(* IEC 61131-3 sources: moqui-plc/simatic-ax/src/moqui/runtime/component/mantle-hvac/src/main/org/moqui/device, 5 files *)

(* ---- AirDistributionControllerStatus.st ---- *)
TYPE AirDistributionControllerStatus : (
    Init,
    HighPhase,
    TransitionToLow,
    LowPhase,
    TransitionToHigh
); END_TYPE

(* ---- DeviceFacade.st ---- *)
(*
 * DeviceFacade implementation for managing devices and logical parameters.
 *
 * Naming rules:
 *   deviceName + parameterName or parameterName -> logical signal
 *   deviceName + parameterName or parameterName + Min/Max -> limits
 *
 * All digital signals (boolean) are active-high (positive logic).
 * All durations are expressed in seconds TUnit.
 *)
TYPE DeviceFacade : STRUCT
	(* HVAC process control parameters (setpoints, limits, etc.) and process sensor signals *)
    (* Cell T+RH sensor  *)
    (* Setpoints and limits - mapped from recipe *)
    tempSetpoint : REAL; (* °C target process temperature *)
    tempHysteresis : REAL; (* °C symmetric hysteresis band *)
    tempMin : REAL;   (* °C absolute lower limit (alarm) *)
    tempMax : REAL; (* °C absolute upper limit (alarm) *)
    rhSetpoint : REAL; (* %  target relative humidity *)
    rhHysteresis : REAL; (* %  symmetric hysteresis band *)
    rhMin : REAL; (* % lower limit *)
    rhMax : REAL; (* % upper limit *)
    (* Feedback - wired from InputSignalUpdate each scan *)
    tempFeedback : REAL; (* °C zone air temperature *)
    rhFeedback : REAL; (* % zone relative humidity *)

    (* Duct T+RH sensor (probe in the pipes) *)
    (* Limits - mapped from recipe or fixed commissioning values *)
    ductTempMin : REAL; (* °C minimum safe supply-air temperature *)
    ductTempMax : REAL; (* °C maximum safe supply-air temperature *)
    ductRhMax : REAL; (* % maximum allowed supply-air humidity *)
    (* Feedback - wired from InputSignalUpdate each scan *)
    ductTempFeedback : REAL; (* °C supply-air temperature in duct *)
    ductRhFeedback : REAL; (* % supply-air relative humidity in duct *)

    (* Boolean predicates - computed each scan by MainRuleEngine *)
    (* Cell sensor *)
    tempInRange : BOOL; (* tempMin+hys <= T <= tempMax-hys *)
    tempAtSetpoint : BOOL; (* |T - Tsp| <= hys *)
    tempAboveSetpointBand : BOOL; (* T >= tempSetpoint + tempHysteresis *)
    tempBelowSetpointBand : BOOL; (* T <= tempSetpoint - tempHysteresis *)
    tempOverMax : BOOL; (* T > tempMax *)
    tempOverMin : BOOL; (* T > tempMin *)
    tempUnderMin : BOOL; (* T < tempMin *)
    tempUnderMax : BOOL; (* T < tempMax *)
    rhAtSetpoint : BOOL;
    rhOverMax  : BOOL; (* RH > rhMax - hys *)
    rhUnderMin : BOOL; (* RH < rhMin + hys *)
    rhOverMin : BOOL;
    rhUnderMax : BOOL;
    (* Duct sensor - safety predicates *)
    ductTempOverMax : BOOL; (* Supply air too hot -> temperature limit violation *)
    ductTempUnderMin : BOOL; (* Supply air too cold -> temperature limit violation *)
    ductRhOverMax : BOOL; (* Supply air saturated -> condensation risk *)

    (* Operating-mode flags and process timing (mapped from recipe). *)
    rhControlEnabled : BOOL; (* Cooling+Heating both active for RH ctrl *)
    rhControlOnly : BOOL; (* Stop when RH <= rhMin regardless of time *)
    (* Air mixing *)
    airMixingEnabled : BOOL;
    airMixingFanEnableRequest : BOOL;
    airMixingFanDisableRequest : BOOL;
    airMixingFan : Actuator;
	(* Air distribution setpoints *)
	airDistributionEnabled : BOOL;
    setPointTimeHigh : UINT; (* Required cumulative time for high throw [s] *)
    setPointTimeLow : UINT; (* Required cumulative time for low throw [s] *)
    (* Process cycle durations (seconds) *)
    processEstimatedDuration : UDINT;
    processMinDuration : UDINT;
    processActualDuration : UDINT;
    processRemainingDuration : UDINT;
    (* Process time tracking *)
    (* Run / break cycle - Mode E *)
    estimatedRuntime : UDINT;
    minRuntime : UDINT;
    actualRuntime : UDINT;
    estimatedBreakDuration : UDINT;
    minBreakDuration : UDINT;
    actualBreakDuration : UDINT;
    (* Flags *)
    timeBreakEnabled : BOOL; (* TRUE while in break period *)
    isCompleted : BOOL; (* TRUE when the work effort is finished *)

    (* Main FSM state and transition request/acknowledge commands *)
    status : MainStatus := MainStatus#Standby;
    lastStatus : MainStatus := MainStatus#Standby;
    (*
     * Internally generated transition requests (set by MainRuleEngine,
     * consumed and cleared by Main.pou each scan)
     *)
    standbyRequest : BOOL;
    ventilationRequest : BOOL;
    coolingRequest : BOOL;
    heatingRequest : BOOL;
    dryingRequest : BOOL;
    faultRequest : BOOL;
    resetRequest : BOOL;

    (* HVAC devices *)

    (* Cold glycol group *)
    (* Enable/disable requests: written by Main component, read by DeviceManager *)
    coldGroupEnableRequest : BOOL;
    coldGroupDisableRequest : BOOL;
    (* Glycol circulating pump - on/off Actuator *)
    coldGlycolPump : Actuator;
    (* Modulating glycol valve - continuous PID control *)
    coldGlycolValve : ProcessPid;

    (* Hot glycol group *)
    hotGroupEnableRequest : BOOL;
    hotGroupDisableRequest : BOOL;
    hotGlycolPump : Actuator;
    hotGlycolValve : ProcessPid;

    (* AHU fan *)
    ahuFanEnableRequest : BOOL;
    (* Speed setpoint (0.0 … 100.0 %) - from recipe *)
    ahuFanSpeedSetpoint : REAL;
    (* Speed feedback (0.0 … 100.0 %) - from InputSignalUpdate *)
    ahuFanSpeedFeedback : REAL;
    ahuFan : ProcessPid;

    (* Air-flow distributor *)
    (* Treated as Actuator with additional ref/feedback.
     * The drive alternates air distribution between left and right ducts.
     * ref = time-split setpoint (0-100 %, 0 = full left, 100 = full right).
     * feedback = actual drive speed feedback.
	 *)
    airFlowEnableRequest : BOOL;
    airFlowDisableRequest : BOOL;
    airFlowRef : REAL; (* duty-cycle / distribution setpoint *)
    airFlowSpeedFeedback : REAL; (* drive speed feedback *)
    airFlow : Actuator;

    (* High flow damper *)
    highFlowDamperEnableRequest : BOOL;
    highFlowDamperDisableRequest : BOOL;
    highFlowDamper : Actuator;

    (* Low flow damper *)
    lowFlowDamperEnableRequest : BOOL;
    lowFlowDamperDisableRequest : BOOL;
    lowFlowDamper : Actuator;

    (* Signal management - centralised fault / alarm / warning engine *)
    signalMgmt : SignalMgmt;
END_STRUCT; END_TYPE

(* ---- AirDistributionController.st ---- *)
(*
 * AirDistributionController: Logical sequencer for alternating high/low air throw.
 *
 * Implements cumulative timing logic for throw phases:
 * - Time advances only during active operation (operationType = Run AND enable = TRUE).
 * - Counters are frozen (retained) during standby/pause phases.
 * - Implements a Make-Before-Break transition between ducts to prevent overpressure peaks,
 * leveraging the asynchronous handshake mechanism (VAR_IN_OUT) of the underlying Actuator instances.
 *)
FUNCTION_BLOCK AirDistributionController
	VAR_EXTERNAL
	    dev : DeviceFacade;
	END_VAR
	VAR_INPUT
	    operationType : OperatingMode := OperatingMode#Init;
	    enable : BOOL; (* Local run permission (e.g., air flow running + air mixing enabled) *)
	    clock1s : BOOL; (* 1-second base clock pulse *)
	END_VAR
	VAR CONSTANT
	    componentName : STRING := 'HVAC_AIR_GROUP';
	END_VAR
	VAR
		(* Logger facade *)
	    logger : LoggerFacade;
	    status : AirDistributionControllerStatus := AirDistributionControllerStatus#Init;
	    cumulatedTimeHigh : UINT := UINT#0;
	    cumulatedTimeLow : UINT := UINT#0;
	END_VAR

	(* Logger facade init *)
	logger.enable := TRUE; logger.loggerName := componentName;

	(* Initialization or reset upon critical Stop *)
	IF operationType = OperatingMode#Init THEN
	    logger(message := 'Init air distribution controller.', level := LogLevel#DEBUG);
	    status := AirDistributionControllerStatus#Init;
	    cumulatedTimeHigh := UINT#0;
	    cumulatedTimeLow := UINT#0;
		dev.highFlowDamperEnableRequest := TRUE;
		dev.highFlowDamperDisableRequest := FALSE;
		dev.lowFlowDamperEnableRequest := FALSE;
		dev.lowFlowDamperDisableRequest := TRUE;
	    RETURN;
	END_IF;

	(* Logic advances ONLY if the system is in Run mode and local enable is active *)
	IF (operationType = OperatingMode#Run) AND enable THEN

	    CASE status OF

	        AirDistributionControllerStatus#Init:
	            (* Startup sequence: defaults to the high throw phase *)
	            dev.highFlowDamperEnableRequest := TRUE;
	 		   	dev.highFlowDamperDisableRequest := FALSE;
	            dev.lowFlowDamperEnableRequest := FALSE;
	 		   	dev.lowFlowDamperDisableRequest := TRUE;
	            logger(message := 'Enter high throw phase.', level := LogLevel#DEBUG);
	            status := AirDistributionControllerStatus#HighPhase;

	        AirDistributionControllerStatus#HighPhase:
	            (* Advance cumulative timer *)
	            IF clock1s THEN
	                cumulatedTimeHigh := cumulatedTimeHigh + UINT#1;
	            END_IF;

	            (* Evaluate switching threshold *)
	            IF dev.setPointTimeHigh > UINT#0 AND cumulatedTimeHigh >= dev.setPointTimeHigh THEN
	                cumulatedTimeHigh := UINT#0;
	                (* Make-Before-Break Interlock / Asynchronous Handshake *)
					dev.highFlowDamperEnableRequest := FALSE;
					dev.highFlowDamperDisableRequest := TRUE;
					dev.lowFlowDamperEnableRequest := TRUE;
					dev.lowFlowDamperDisableRequest := FALSE;
	                logger(message := 'Transition to low throw.', level := LogLevel#DEBUG);
	                status := AirDistributionControllerStatus#TransitionToLow;
	            END_IF;

	        AirDistributionControllerStatus#TransitionToLow:
	            (* * Monitor the falling edge of the request signals.
	             * The Actuator block internally clears the VAR_IN_OUT variable once
	             * the physical maneuver is completed. This ensures the sequencer
	             * advances only after the hardware has reached its target position.
	             *)
	            IF NOT dev.highFlowDamperDisableRequest AND NOT dev.lowFlowDamperEnableRequest THEN
	                logger(message := 'Enter low throw phase.', level := LogLevel#DEBUG);
	                status := AirDistributionControllerStatus#LowPhase;
	            END_IF;

	        AirDistributionControllerStatus#LowPhase:
	            (* Advance cumulative timer *)
	            IF clock1s THEN
	                cumulatedTimeLow := cumulatedTimeLow + UINT#1;
	            END_IF;

	            (* Evaluate switching threshold *)
	            IF dev.setPointTimeLow > UINT#0 AND cumulatedTimeLow >= dev.setPointTimeLow THEN
	                cumulatedTimeLow := UINT#0;
	                (* Make-Before-Break Interlock / Asynchronous Handshake *)
					dev.highFlowDamperEnableRequest := TRUE;
					dev.highFlowDamperDisableRequest := FALSE;
					dev.lowFlowDamperEnableRequest := FALSE;
					dev.lowFlowDamperDisableRequest := TRUE;
	                logger(message := 'Transition to high throw.', level := LogLevel#DEBUG);
	                status := AirDistributionControllerStatus#TransitionToHigh;
	            END_IF;

	        AirDistributionControllerStatus#TransitionToHigh:
	            (* Wait for hardware positioning confirmation *)
	            IF NOT dev.lowFlowDamperDisableRequest AND NOT dev.highFlowDamperEnableRequest THEN
	                logger(message := 'Enter high throw phase.', level := LogLevel#DEBUG);
	                status := AirDistributionControllerStatus#HighPhase;
	            END_IF;
	    END_CASE;
	ELSE
	    (* Standby / Pause Condition *)
	    (*
	     * During standby (OperatingMode#Standby OR enable = FALSE), the FB does
	     * not increment any timers. The current status and Request variables are
	     * frozen, maintaining the hardware in its last consolidated stable state.
	     *)
	    ;
	END_IF;
	END_FUNCTION_BLOCK

(* ---- DeviceDiagnostics.st ---- *)
(* Device diagnostics *)
FUNCTION_BLOCK DeviceDiagnostics
	VAR_EXTERNAL
		dev : DeviceFacade;
	END_VAR
	VAR_INPUT
		operationType : OperatingMode := OperatingMode#Run;
	END_VAR
	VAR_OUTPUT
		error : BOOL;
	END_VAR

	error := TRUE;

	(* Signal management engine *)
	(*
	 * Prepare a fresh scan (clears the accumulated output action).
	 * Then process each device signal in priority order.
	 * ImmediateStop -> faultRequest := TRUE -> Main enters Fault state.
	 *)
	dev.signalMgmt(operationType := SignalMgmtOperatingMode#Prepare);
	dev.signalMgmt.operationType := SignalMgmtOperatingMode#Process;

	(* Device faults *)
	dev.signalMgmt(
		loggerName := dev.ahuFan.loggerName,
		code := 16#0001,
		category := SignalCategory#Alarm,
		resetPol := ResetPolicy#UnconditionedReset,
		activationCondition := dev.ahuFan.invalidConfig,
		outputAction := DWORD#16#0002);
	dev.signalMgmt(
		loggerName := dev.airFlow.loggerName,
		code := 16#0002,
		category := SignalCategory#Alarm,
		resetPol := ResetPolicy#UnconditionedReset,
		activationCondition := dev.airFlow.fault,
		outputAction := DWORD#16#0002);
	dev.signalMgmt(
		loggerName := dev.coldGlycolPump.loggerName,
		code := 16#0003,
		category := SignalCategory#Alarm,
		resetPol := ResetPolicy#UnconditionedReset,
		activationCondition := dev.coldGlycolPump.fault,
		outputAction := DWORD#16#0002);
	dev.signalMgmt(
		loggerName := dev.coldGlycolValve.loggerName,
		code := 16#0004,
		category := SignalCategory#Alarm,
		resetPol := ResetPolicy#UnconditionedReset,
		activationCondition := dev.coldGlycolValve.invalidConfig,
		outputAction := DWORD#16#0002);
	dev.signalMgmt(
		loggerName := dev.hotGlycolPump.loggerName,
		code := 16#0005,
		category := SignalCategory#Alarm,
		resetPol := ResetPolicy#UnconditionedReset,
		activationCondition := dev.hotGlycolPump.fault,
		outputAction := DWORD#16#0002);
	dev.signalMgmt(
		loggerName := dev.hotGlycolValve.loggerName,
		code := 16#0006,
		category := SignalCategory#Alarm,
		resetPol := ResetPolicy#UnconditionedReset,
		activationCondition := dev.hotGlycolValve.invalidConfig,
		outputAction := DWORD#16#0002);
	dev.signalMgmt(
		loggerName := dev.highFlowDamper.loggerName,
		code := 16#0007,
		category := SignalCategory#Alarm,
		resetPol := ResetPolicy#UnconditionedReset,
		activationCondition := dev.highFlowDamper.fault,
		outputAction := DWORD#16#0002);
	dev.signalMgmt(
		loggerName := dev.lowFlowDamper.loggerName,
		code := 16#0008,
		category := SignalCategory#Alarm,
		resetPol := ResetPolicy#UnconditionedReset,
		activationCondition := dev.lowFlowDamper.fault,
		outputAction := DWORD#16#0002);

	(*
	 * Duct safety alarms - supply-air temperature limits (ImmediateStop).
	 * Air that is too hot or too cold entering the curing room can damage
	 * or contaminate the product. These alarms are always evaluated
	 * regardless of the current FSM state.
	 *)
	dev.signalMgmt(
		loggerName := 'HVAC_DEMO_PLC',
		code := 16#0010,
		category := SignalCategory#Alarm,
		resetPol := ResetPolicy#UnconditionedReset,
		activationCondition := dev.ductTempOverMax,
		outputAction := DWORD#16#0002);
	dev.signalMgmt(
		loggerName := 'HVAC_DEMO_PLC',
		code := 16#0011,
		category := SignalCategory#Alarm,
		resetPol := ResetPolicy#UnconditionedReset,
		activationCondition := dev.ductTempUnderMin,
		outputAction := DWORD#16#0002);

	(* Duct RH - Warning only (condensation risk, does not stop the machine) *)
	dev.signalMgmt(
		loggerName := 'HVAC_DEMO_PLC',
		code := 16#0012,
		category := SignalCategory#Warning,
		resetPol := ResetPolicy#UnconditionedReset,
		activationCondition := dev.ductRhOverMax,
		outputAction := DWORD#16#0000);

	error := FALSE;
	END_FUNCTION_BLOCK

(* ---- DeviceManager.st ---- *)
(* Hardware Abstraction Layer (HAL) orchestrator.
 *
 * Drives all physical device FBs once per scan.
 * Main component sets the enable/disable request flags; DeviceManager wires them
 * to the individual Actuator / ProcessPid FBs.
 *
 * Call order within the PLC task:
 *   InputSignalUpdate (updates feedback signals from field)
 *   Main (FSM + MainRuleEngine -> sets request flags)
 *   DeviceManager (this block - drives device FBs)
 *   OutputSignalUpdate (maps device outputs to physical terminals)
 *
 * Handshake note (Actuator FBs):
 *   enableRequest / disableRequest are VAR_IN_OUT.  The Actuator FB clears
 *   the flag as its acknowledgment.  Main.pou re-asserts the flag each scan
 *   from dev.xxxEnableRequest, so the handshake is level-triggered.
 *
 * ProcessPid note (ahuFan):
 *   ProcessPid uses a plain BOOL 'enable' input - no VAR_IN_OUT handshake.
 *   Setting enable := FALSE ramps the output to 0 and disables the controller.
 *)
FUNCTION_BLOCK DeviceManager
	VAR_EXTERNAL
		clks : Clocks;
		dev : DeviceFacade;
	END_VAR
	VAR_INPUT
		operationType : OperatingMode := OperatingMode#Run;
	END_VAR

	(* Cold glycol group *)
	(*
	 * Pump is started first via the request/ack handshake.
	 * Valve enable follows the group request directly (no separate handshake
	 * needed for ProcessPid - enable := FALSE freezes the output at 0).
	 *)
	dev.coldGlycolPump(
		operationType := operationType,
		clock := clks.clock100ms,
		enableRequest := dev.coldGroupEnableRequest,
		disableRequest := dev.coldGroupDisableRequest);

	dev.coldGlycolValve(
		enable := dev.coldGroupEnableRequest,
		feedback := dev.tempFeedback,
		setpoint := dev.tempSetpoint,
		clock := clks.clock100ms);

	(* Hot glycol group *)
	dev.hotGlycolPump(
		operationType := operationType,
		clock := clks.clock100ms,
		enableRequest := dev.hotGroupEnableRequest,
		disableRequest := dev.hotGroupDisableRequest);

	dev.hotGlycolValve(
		enable := dev.hotGroupEnableRequest,
		feedback := dev.tempFeedback,
		setpoint := dev.tempSetpoint,
		clock := clks.clock100ms);

	(* AHU fan *)
	(*
	 * enable := FALSE ramps down the drive and disables the PID output.
	 * Speed setpoint (ahuFanSpeedSetpoint) and the PID tuning parameters
	 * (gain, integrationTime, etc.) are mapped from the device config (recipe).
	 * ahuFanSpeedFeedback is wired from InputSignalUpdate (drive feedback word).
	 *)
	dev.ahuFan(
		enable := dev.ahuFanEnableRequest,
		setpoint := dev.ahuFanSpeedSetpoint,
		feedback := dev.ahuFanSpeedFeedback,
		clock := clks.clock100ms);

	(* Air flow distributor (drive) *)
	(*
	 * Treated as Actuator with an additional speed reference.
	 * ref = distribution setpoint (0-100 %) from device config (recipe)/RuleEngine.
	 * feedback = drive speed feedback from InputSignalUpdate.
	 * The drive alternates supply air between left and right ducts
	 * according to the ref timing programmed on the drive itself;
	 * the PLC only starts / stops it and adjusts the reference level.
	 *)
	dev.airFlow(
		operationType := operationType,
		clock := clks.clock100ms,
		enableRequest := dev.airFlowEnableRequest,
		disableRequest := dev.airFlowDisableRequest,
		referenceValue := dev.airFlowRef,
		feedback := dev.airFlowSpeedFeedback);

	(* High Flow Damper *)
	(* Requests are generated by AirDistributionController when air mixing is enabled. *)
	dev.highFlowDamper(
		operationType := operationType,
		clock := clks.clock100ms,
		enableRequest := dev.highFlowDamperEnableRequest,
		disableRequest := dev.highFlowDamperDisableRequest);

	(* Low Flow Damper *)
	(* Requests are generated by AirDistributionController when air mixing is enabled. *)
	dev.lowFlowDamper(
		operationType := operationType,
		clock := clks.clock100ms,
		enableRequest := dev.lowFlowDamperEnableRequest,
		disableRequest := dev.lowFlowDamperDisableRequest);
	END_FUNCTION_BLOCK
